(**************************************************************************************
 * 	Application		:	BoxControl Framework
 *	Revision		:	$Revision: 404529 $
 *	Revision date	:	$Date: 2018-04-23 08:21:38 +0200 (Mo., 23 Apr 2018) $
 *	Last changed by	:	$Author: b7bolm $
 *	URL				:	$URL: http://almscdc.swisslog.com/repo/SWPD/Development/BoxControlFramework/20_Release/trunk/01_Software/BCF/BCF/JumpStart/20_Product/10_App/10_Base/10_Lib/00_GVLs/ISR_Table.TcGVL $
 *
 *	Purpose			:	ISR signals - Separated due to debug reasons.
 *
 * ------------------------------------------------------------------------------------
 *	Copyright Swisslog [IP AG], Switzerland. All rights reserved.
 * 
 * ------------------------------------------------------------------------------------
 *	
 * 	Revision History: 
 *
 * 	VERSION			DATE			INITIALS			DESCRIPTION
 *	0.1				01.01.2001		swl					Example
 *
 **************************************************************************************)

VAR_GLOBAL CONSTANT
	NUMBER_OF_ISR_SIGNALS			: INT := 9999; // Number of ISR signals, max 9999 
	NUMBER_OF_ISR_DATA_LENGTH		: INT := 99; // Max length of data
END_VAR
 
VAR_GLOBAL
	ISR_SignalType					: ARRAY [0..2] OF ST_ISR_Table;	
END_VAR

(* stored: Version 1.1.0.1, ProductVersion 3.1.4022.12
   GVL ISR_Table: Id {9d336346-99ca-4cf9-9ba3-0bb28b2cc0cb} *)
